{attribute 'linkalways'} 
{attribute 'no_explicit_call' := 'This FB is a CLASS and must be accessed using methods or properties'}
{attribute 'enable_dynamic_creation'}
FUNCTION_BLOCK MoveAdditiveCommand EXTENDS Mc2AsyncCommand
VAR
	fb : Tc2_Mc2.Mc_MoveAdditive;
END_VAR

{attribute 'monitoring' := 'call'}
PROPERTY PUBLIC Active : BOOL
GET // PUBLIC
Active := fb.Active;
END_GET
END_PROPERTY

METHOD PUBLIC CyclicCall
SUPER^.CyclicCall();
fb(Axis := axis_ref);
END_METHOD

(*FB_Init is always available implicitly and it is used primarily for initialization.
The return value is not evaluated. For a specific influence, you can also declare the
methods explicitly and provide additional code there with the standard initialization
code. You can evaluate the return value.*)
METHOD FB_Init : BOOL
VAR_INPUT
	(* TRUE: the retain variables are initialized (reset warm / reset cold)*)
	bInitRetains : BOOL;
	(* TRUE: the instance will be copied to the copy code afterward (online change)*)
	bInCopyCode	: BOOL;
	axis : REFERENCE TO Mc2Axis;
	velocity : LREAL;
	acceleration : LREAL := 0;
	deceleration : LREAL := 0;
	jerk : LREAL := 0;
	buffer_mode	: MotionBufferMode := MotionBufferMode.Aborting;
END_VAR
fb.Velocity := velocity;
fb.Acceleration := acceleration;
fb.Deceleration := deceleration;
fb.Jerk := jerk;
fb.BufferMode := Mc2BufferModeConvertTo(buffer_mode);
END_METHOD

METHOD PROTECTED OnExecuting
VAR_INPUT
	state_control : AsyncCommandStateControl;
END_VAR
fb.Execute := TRUE;

IF fb.Done THEN
	state_control.Next();
	fb.Execute := FALSE;
END_IF

IF fb.CommandAborted THEN
	Abort();
	fb.Execute := FALSE;
END_IF

IF fb.Error THEN
	state_control.Error(fb.ErrorId);
	fb.Execute := FALSE;
END_IF
END_METHOD

END_FUNCTION_BLOCK

(* stored: Version 1.1.0.1, ProductVersion 3.1.4026.13
   POU MoveAdditiveCommand: Id {42f22a6c-7a89-42c4-8079-dce57b8029da}, SpecialFunc None
   Property Active: Id {06662ea0-4a5f-4fe8-acb9-0a896ee25b75}
   Get Get: Id {57a3d9c6-3d75-4db5-988f-0ed9f570875d}
   Method CyclicCall: Id {d970fcd9-ce09-46ba-9e85-ecda5668d725}
   Method FB_Init: Id {01fc868d-8bc5-4ddd-8112-8565f6337198}
   Method OnExecuting: Id {f03cd200-84fb-4dcb-8ae7-ebeb1c89b675} *)
